(* IEC 61131-3 sources: AI_PLC/motion_stubs, 7 files *)

(* ---- AxisTypes.st ---- *)
(* Virtual axis simulation model shared by all MC_* stub function blocks.
   AxisState values: 0=Disabled 1=Standstill 2=Homing 3=DiscreteMotion 4=ContinuousMotion 5=Stopping 6=ErrorStop
   ErrorID values: 1=EStop 2=LimitSwitch *)

TYPE AXIS_REF :
STRUCT
    Position        : REAL;
    Velocity        : REAL;
    TargetPosition  : REAL;
    TargetVelocity  : REAL;
    Accel           : REAL;
    Decel           : REAL;
    Direction       : INT;
    CommandId       : DINT;
    AxisState       : INT;
    Enabled         : BOOL;
    Homed           : BOOL;
    Busy            : BOOL;
    Done            : BOOL;
    Active          : BOOL;
    CommandAborted  : BOOL;
    Error           : BOOL;
    ErrorID         : DINT;
    InVelocity      : BOOL;
    EStopActive     : BOOL;
    LimitPos        : BOOL;
    LimitNeg        : BOOL;
    HomeSwitch      : BOOL;
END_STRUCT;
END_TYPE

(* Fixed simulated scan period (seconds), inlined as a literal in each FB below
   rather than a shared VAR_GLOBAL -- this matiec build rejects VAR_GLOBAL
   declared outside a CONFIGURATION/RESOURCE. Scenario assertions must be
   scan-count/state-based, never wall-clock-based, so the exact value here
   only affects how many scans a move takes, not correctness. *)

(* ---- MC_Home.st ---- *)
FUNCTION_BLOCK MC_Home
VAR_INPUT
    Execute  : BOOL;
    Velocity : REAL;
END_VAR
VAR_OUTPUT
    Done  : BOOL;
    Busy  : BOOL;
    Error : BOOL;
END_VAR
VAR_IN_OUT
    Axis : AXIS_REF;
END_VAR
VAR
    execRise : R_TRIG;
    active   : BOOL;
END_VAR

execRise(CLK := Execute);

IF execRise.Q AND NOT active THEN
    IF NOT Axis.Enabled OR Axis.EStopActive THEN
        Error := TRUE;
    ELSE
        active := TRUE;
        Axis.Busy := TRUE;
        Axis.Done := FALSE;
        Axis.Homed := FALSE;
        Axis.AxisState := 2;
        Error := FALSE;
    END_IF;
END_IF;

IF active THEN
    IF Axis.EStopActive THEN
        Axis.Velocity := 0.0;
        Axis.Busy := FALSE;
        Axis.Error := TRUE;
        Axis.ErrorID := 1;
        Axis.AxisState := 6;
        active := FALSE;
        Error := TRUE;
    ELSIF Axis.HomeSwitch OR Axis.LimitNeg THEN
        Axis.Velocity := 0.0;
        Axis.Position := 0.0;
        Axis.Homed := TRUE;
        Axis.Done := TRUE;
        Axis.Busy := FALSE;
        Axis.AxisState := 1;
        active := FALSE;
    ELSE
        Axis.Velocity := Velocity;
        Axis.Position := Axis.Position - Velocity * 0.01;
    END_IF;
END_IF;

Busy := active;
Done := Axis.Homed AND NOT active;

END_FUNCTION_BLOCK

(* ---- MC_MoveAbsolute.st ---- *)
FUNCTION_BLOCK MC_MoveAbsolute
VAR_INPUT
    Execute  : BOOL;
    Position : REAL;
    Velocity : REAL;
END_VAR
VAR_OUTPUT
    Done           : BOOL;
    Busy           : BOOL;
    Active         : BOOL;
    CommandAborted : BOOL;
    Error          : BOOL;
END_VAR
VAR_IN_OUT
    Axis : AXIS_REF;
END_VAR
VAR
    execRise  : R_TRIG;
    execFall  : F_TRIG;
    myCommand : DINT;
    owned     : BOOL;
END_VAR

execRise(CLK := Execute);
execFall(CLK := Execute);

IF execRise.Q THEN
    IF NOT Axis.Enabled OR Axis.EStopActive OR Axis.AxisState = 6 THEN
        CommandAborted := TRUE;
        Error := TRUE;
    ELSIF Axis.Busy AND Axis.CommandId <> myCommand THEN
        CommandAborted := TRUE;
        Error := TRUE;
    ELSE
        Axis.CommandId := Axis.CommandId + 1;
        myCommand := Axis.CommandId;
        owned := TRUE;
        Axis.TargetPosition := Position;
        Axis.TargetVelocity := Velocity;
        Axis.Busy := TRUE;
        Axis.Active := TRUE;
        Axis.Done := FALSE;
        Axis.AxisState := 3;
        CommandAborted := FALSE;
        Error := FALSE;
    END_IF;
END_IF;

IF owned AND Axis.CommandId = myCommand THEN
    IF Axis.EStopActive THEN
        Axis.Velocity := 0.0;
        Axis.Busy := FALSE;
        Axis.Active := FALSE;
        Axis.Error := TRUE;
        Axis.ErrorID := 1;
        Axis.AxisState := 6;
        CommandAborted := TRUE;
        owned := FALSE;
    ELSIF (Axis.TargetPosition > Axis.Position AND Axis.LimitPos) OR
          (Axis.TargetPosition < Axis.Position AND Axis.LimitNeg) THEN
        Axis.Velocity := 0.0;
        Axis.Busy := FALSE;
        Axis.Active := FALSE;
        Axis.Error := TRUE;
        Axis.ErrorID := 2;
        Axis.AxisState := 6;
        CommandAborted := TRUE;
        owned := FALSE;
    ELSE
        Axis.Velocity := Axis.TargetVelocity;
        IF Axis.TargetPosition > Axis.Position THEN
            Axis.Position := Axis.Position + Axis.Velocity * 0.01;
            IF Axis.Position >= Axis.TargetPosition THEN
                Axis.Position := Axis.TargetPosition;
            END_IF;
        ELSE
            Axis.Position := Axis.Position - Axis.Velocity * 0.01;
            IF Axis.Position <= Axis.TargetPosition THEN
                Axis.Position := Axis.TargetPosition;
            END_IF;
        END_IF;

        IF Axis.Position = Axis.TargetPosition THEN
            Axis.Velocity := 0.0;
            Axis.Busy := FALSE;
            Axis.Active := FALSE;
            Axis.Done := TRUE;
            Axis.AxisState := 1;
        END_IF;
    END_IF;
END_IF;

Busy := owned AND Axis.Busy;
Active := owned AND Axis.Active;
Done := owned AND Axis.Done;

IF execFall.Q THEN
    Axis.Done := FALSE;
    owned := FALSE;
END_IF;

END_FUNCTION_BLOCK

(* ---- MC_MoveVelocity.st ---- *)
FUNCTION_BLOCK MC_MoveVelocity
VAR_INPUT
    Execute      : BOOL;
    Velocity     : REAL;
    Acceleration : REAL;
END_VAR
VAR_OUTPUT
    InVelocity     : BOOL;
    Busy           : BOOL;
    Active         : BOOL;
    CommandAborted : BOOL;
    Error          : BOOL;
END_VAR
VAR_IN_OUT
    Axis : AXIS_REF;
END_VAR
VAR
    myCommand : DINT;
    owned     : BOOL;
END_VAR

IF Execute THEN
    IF NOT owned THEN
        IF NOT Axis.Enabled OR Axis.EStopActive OR Axis.AxisState = 6 THEN
            CommandAborted := TRUE;
            Error := TRUE;
        ELSIF Axis.Busy AND Axis.CommandId <> myCommand THEN
            CommandAborted := TRUE;
            Error := TRUE;
        ELSE
            Axis.CommandId := Axis.CommandId + 1;
            myCommand := Axis.CommandId;
            owned := TRUE;
            Axis.TargetVelocity := Velocity;
            Axis.Active := TRUE;
            Axis.AxisState := 4;
            CommandAborted := FALSE;
            Error := FALSE;
        END_IF;
    END_IF;

    IF owned AND Axis.CommandId = myCommand THEN
        IF Axis.EStopActive THEN
            Axis.Velocity := 0.0;
            Axis.Active := FALSE;
            Axis.InVelocity := FALSE;
            Axis.Error := TRUE;
            Axis.ErrorID := 1;
            Axis.AxisState := 6;
            CommandAborted := TRUE;
            owned := FALSE;
        ELSE
            IF Axis.Velocity < Velocity THEN
                Axis.Velocity := Axis.Velocity + Acceleration * 0.01;
                IF Axis.Velocity >= Velocity THEN
                    Axis.Velocity := Velocity;
                END_IF;
            ELSIF Axis.Velocity > Velocity THEN
                Axis.Velocity := Axis.Velocity - Acceleration * 0.01;
                IF Axis.Velocity <= Velocity THEN
                    Axis.Velocity := Velocity;
                END_IF;
            END_IF;

            IF Axis.Velocity = Velocity THEN
                InVelocity := TRUE;
                Axis.InVelocity := TRUE;
            ELSE
                InVelocity := FALSE;
                Axis.InVelocity := FALSE;
            END_IF;

            IF Velocity >= 0.0 THEN
                Axis.Position := Axis.Position + Axis.Velocity * 0.01;
            ELSE
                Axis.Position := Axis.Position - Axis.Velocity * 0.01;
            END_IF;
        END_IF;
    END_IF;
ELSE
    IF owned THEN
        Axis.Active := FALSE;
        Axis.AxisState := 1;
        Axis.InVelocity := FALSE;
        owned := FALSE;
    END_IF;
    InVelocity := FALSE;
END_IF;

Busy := owned;
Active := owned AND Axis.Active;

END_FUNCTION_BLOCK

(* ---- MC_Power.st ---- *)
FUNCTION_BLOCK MC_Power
VAR_INPUT
    Enable : BOOL;
END_VAR
VAR_OUTPUT
    Status : BOOL;
    Error  : BOOL;
END_VAR
VAR_IN_OUT
    Axis : AXIS_REF;
END_VAR

IF Axis.EStopActive THEN
    Axis.Enabled := FALSE;
ELSIF Enable AND Axis.AxisState <> 6 THEN
    Axis.Enabled := TRUE;
ELSE
    Axis.Enabled := FALSE;
END_IF;

IF Axis.AxisState = 0 AND Axis.Enabled THEN
    Axis.AxisState := 1;
END_IF;
IF NOT Axis.Enabled AND Axis.AxisState <> 6 THEN
    Axis.AxisState := 0;
END_IF;

Status := Axis.Enabled;
Error := Axis.Error;

END_FUNCTION_BLOCK

(* ---- MC_Reset.st ---- *)
FUNCTION_BLOCK MC_Reset
VAR_INPUT
    Execute : BOOL;
END_VAR
VAR_OUTPUT
    Done  : BOOL;
    Error : BOOL;
END_VAR
VAR_IN_OUT
    Axis : AXIS_REF;
END_VAR
VAR
    prevExecute : BOOL;
END_VAR

IF Execute AND NOT prevExecute THEN
    IF NOT Axis.EStopActive THEN
        Axis.Error := FALSE;
        Axis.ErrorID := 0;
        Axis.CommandAborted := FALSE;
        IF Axis.AxisState = 6 THEN
            Axis.AxisState := 1;
        END_IF;
        Done := TRUE;
    ELSE
        Done := FALSE;
    END_IF;
ELSE
    Done := FALSE;
END_IF;
prevExecute := Execute;
Error := Axis.Error;

END_FUNCTION_BLOCK

(* ---- MC_Stop.st ---- *)
FUNCTION_BLOCK MC_Stop
VAR_INPUT
    Execute      : BOOL;
    Deceleration : REAL;
END_VAR
VAR_OUTPUT
    Done : BOOL;
    Busy : BOOL;
END_VAR
VAR_IN_OUT
    Axis : AXIS_REF;
END_VAR
VAR
    active : BOOL;
END_VAR

IF Execute THEN
    active := TRUE;
END_IF;

IF active THEN
    Axis.AxisState := 5;
    Axis.Busy := TRUE;
    IF Axis.Velocity > 0.0 THEN
        Axis.Velocity := Axis.Velocity - Deceleration * 0.01;
        IF Axis.Velocity <= 0.0 THEN
            Axis.Velocity := 0.0;
        END_IF;
    ELSIF Axis.Velocity < 0.0 THEN
        Axis.Velocity := Axis.Velocity + Deceleration * 0.01;
        IF Axis.Velocity >= 0.0 THEN
            Axis.Velocity := 0.0;
        END_IF;
    END_IF;

    IF Axis.Velocity = 0.0 THEN
        Done := TRUE;
        Axis.Busy := FALSE;
        Axis.Active := FALSE;
        Busy := FALSE;
        IF NOT Execute THEN
            active := FALSE;
            IF Axis.AxisState = 5 THEN
                Axis.AxisState := 1;
            END_IF;
        END_IF;
    ELSE
        Done := FALSE;
        Busy := TRUE;
    END_IF;
ELSE
    Done := FALSE;
    Busy := FALSE;
END_IF;

END_FUNCTION_BLOCK
